PROGRAM TEST
VAR
// create an instance for all FB in base project in order to test if there are errors in the FB ()

	moyenne_test : MOYENNE;
	time_Test : TIME := T#5s;
	bTest : BOOL;
	rValue : REAL;
	
END_VAR


moyenne_test(
	In_fenetre_mesure := time_Test,
	In_synchro := CalLocalTimeStruct.wSecond MOD 5 = 0,
	In_valeur := word_to_real(CalLocalTimeStruct.wSecond)
);
moyenne_test.Calcul();

END_PROGRAM

(* stored: Version 1.1.0.1, ProductVersion 3.1.4024.11
   POU TEST: Id {a4afb91a-1cb7-4580-848e-d5f5a964dc59}, SpecialFunc None *)
